// TIA Portal V20 export
// export: Created 2025-12-01T14:57:20.1879597Z, ExportSetting None, DisplayName Totally Integrated Automation Portal, DisplayVersion V20 Update 3, DisplayName TIA Portal Openness, DisplayVersion V20 Update 3, DisplayName TIA Portal Version Control Interface, DisplayVersion V20 Update 3, DisplayName STEP 7 Professional, DisplayVersion V20 Update 3, DisplayName STEP 7 Safety, DisplayVersion V20 Update 2, DisplayName WinCC Basic/Comfort/Advanced, DisplayVersion V20 Update 3, DisplayName WinCC Professional, DisplayVersion V20 Update 3, DisplayName WinCC Unified, DisplayVersion V20 Update 3
DATA_BLOCK "DB906_Interlocks"   // DB906
{ S7_Optimized_Access := 'FALSE'; DB_Accessible_From_OPC_UA := 'FALSE' }
// stored: AutoNumber false, DBAccessibleFromOPCUA false
   VAR
      Interlock { S7_SetPoint := 'True'} : Array[1.."CTE_MaxMesas"] of "UDT_Interlock_generico";
      Interlock_manual { S7_SetPoint := 'True'} : Array[1.."CTE_MaxMesas"] of "UDT_Interlock_manual";
   END_VAR
BEGIN
END_DATA_BLOCK
